  //-------------------------------------------------------------------------------------------------
  // XTS Environment; ProcessingUnit, Part, Track, Mover
  //  - instances are initialized by getting OTCIDs
  //-------------------------------------------------------------------------------------------------
  _nXpu                       : UINT := 1;  // input property in case of multiple XPU in project
  _nGroup                     : UINT;       // input property in case of multiple Xpu in project

  _nTrack                     : UINT := 1;  // this example is intended for one track only

  {attribute 'displaymode':='hex'}
  _CaGroupOID                 : OTCID; // input property frome cyclic CA group interface, MUST be set in order to do successful INIT

  // checked and evaluated in XpuCheckCycle()
  _bAllPositionsValid,
  _bMoverIdDetectionValid,
  _bMoverIdDetectionError     : BOOL;

  _nDetectedMoverCount,
  _nExpectedMoverCount        : UINT;

  _XpuOperationMode           : OperationMode;
  _MoverIdDetectionMode       : MoverIdDetectionMode;

  // XTS_Utility connection to TcCOM Object
  _fbEnvironment              : Tc3_XTS_Utility.FB_TcIoXtsEnvironment;

  // local instances of members of Environment
  // local members are connected to TcCOM by XpuInit()
  _fbProcessingUnit           : Tc3_XTS_Utility.FB_TcIoXtsProcessingUnit;

  _fbXpuPart                  : Tc3_XTS_Utility.FB_TcIoXtsXpuPart;
  _fbXpuTrack                 : Tc3_XTS_Utility.FB_TcIoXtsXpuTrack;

  _fbMc2CaGroup               : Tc3_XTS_Utility.FB_Mc2CaGroup;

  _fbPartModules              : ARRAY[1..MAX_MODULE]  OF Tc3_XTS_Utility.FB_TcIoXtsPartModule;
  _fbMoverXpu                 : ARRAY[1..MAX_MOVER]   OF Tc3_XTS_Utility.FB_TcIoXtsXpuMover;

  // TcCOM ObjectId (who am I talking to?)
  {attribute 'displaymode':='hex'}
  _Xpu_OTCID                  : OTCID;
  {attribute 'displaymode':='hex'}
  _Group_OTCID                : ARRAY[1..MAX_GROUP]   OF OTCID; // OTCID read from XPU
  {attribute 'displaymode':='hex'}
  _Part_OTCID                 : ARRAY[1..MAX_PART]    OF OTCID;
  {attribute 'displaymode':='hex'}
  _Track_OTCID                : ARRAY[1..MAX_TRACK]   OF OTCID;
  {attribute 'displaymode':='hex'}
  _Mov_OTCID                  : ARRAY[1..MAX_MOVER]   OF OTCID;
  {attribute 'displaymode':='hex'}
  _Module_OTCID               : ARRAY[1..MAX_MODULE]  OF OTCID;

  // COE Data access
  _ModuleInfoData             : REFERENCE TO ARRAY[1..MAX_MODULE] OF Tc3_XTS_Utility.ST_InfoDataView;
  _bModulePower               : ARRAY[1..MAX_MODULE] OF BOOL;

  // double check RailLength, XpuInit() will get stuck in error if not configured correctly
  _RailLengthXpu              : LREAL;
  _RailLengthGroup            : LREAL;

  _nLengthXpu,
  _nLengthGroup               : UINT;

  _nInfoServerCount,
  _nIfoStationCount,
  _nPartCount,
  _nTrackCount,
  _nTaskCount,
  _nMoverCount,
  _nModuleCount,
  _nCheckMovOID,
  _nCheckModAdr               : UINT;

  _ix                         : UINT;

  {attribute 'hide'}
  _XpuInfo                    : ST_XPU_INFO;
END_VAR

// get DcLink information from motor modules
PROPERTY AllModulesDcLink : bool
GET
VAR
  _bTmp     : BOOL;
  _nModule  : UINT;
END_VAR
IF NOT (_eInit = E_XPU_INIT.INIT_DONE) THEN RETURN; END_IF

FOR _nModule := 1 TO _nModuleCount
DO
  IF NOT _bModulePower[_nModule] // information comes from cyclic call in Cycle(): ModuleInfoData()
  THEN
    _bTmp  := FALSE;
    EXIT;
  ELSE
    _bTmp  := TRUE;
  END_IF
END_FOR

AllModulesDcLink := _bTmp;
END_GET
END_PROPERTY

PROPERTY CaGroupOID : OTCID
SET
// Group OTCID must come from the CA Group mapping in NC.Objects
_CaGroupOID := CaGroupOID;
END_SET
END_PROPERTY

METHOD Cycle : E_PROGRESS
VAR_INPUT
  Enable      : BOOL; // enable to do cyclic checks on Environment and its members
END_VAR
VAR_IN_OUT
  _eChk       : E_XPU_CHECK;
END_VAR
VAR_INST

  _eJobResult,
  _eResult      : E_PROGRESS;
  _eState       : E_PROGRESS := E_PROGRESS.PROGRESS_INIT;

END_VAR
IF NOT Enable
THEN
  ModuleInfoData(FALSE);

  _eResult  :=
  _eState   := E_PROGRESS.PROGRESS_INIT; 
  _eChk     := E_XPU_CHECK.INIT_CHECK;
END_IF 
//-----------------------------------------------------------------------------
// cyclic data fetch from Environment, ProcessingUnit, Part, ...
//-----------------------------------------------------------------------------
CASE _eState
OF
  E_PROGRESS.PROGRESS_INIT:
    IF Enable
    THEN
      _eState := _eResult         := E_PROGRESS.PROGRESS_BUSY;
    END_IF

  //---------------------------------------------------------------------------
  E_PROGRESS.PROGRESS_BUSY:       // get data from Xpu, ProcessingUnit, Part, XpuCaGroup
    _eState                       := E_PROGRESS.PROGRESS_STARTUP;

    _bAllPositionsValid           := _fbProcessingUnit.GetAreAllPositionsValid();
    _nDetectedMoverCount          := TO_UINT(_fbProcessingUnit.GetDetectedMoverCount());
    _nExpectedMoverCount          := TO_UINT(_fbProcessingUnit.GetExpectedMoverCount());
  
    _XpuOperationMode             := _fbProcessingUnit.GetOperationMode();
    _MoverIdDetectionMode         := _fbProcessingUnit.GetMoverIdDetectionMode();
  
    _RailLengthXpu                := _fbXpuPart.GetLength();
    _RailLengthGroup              := _fbMc2CaGroup.GetRailLength();
    _nLengthXpu                   := TO_UINT(_RailLengthXpu);
    _nLengthGroup                 := TO_UINT(_RailLengthGroup);
END_CASE
//-----------------------------------------------------------------------------
//-----------------------------------------------------------------------------
CASE _eState
OF
  //---------------------------------------------------------------------------
  E_PROGRESS.PROGRESS_STARTUP:    // check data for errors
    IF NOT (_bAllPositionsValid)
    THEN
      _bAllPositionsValid         := FALSE;
      _eChk                       := E_XPU_CHECK.PROCESSING_UNIT_POSITIONS_VALID;
      _eState := _eResult         := E_PROGRESS.PROGRESS_ERROR;

    ELSIF NOT (_nLengthXpu > 0)
    THEN
      _eChk                       := E_XPU_CHECK.XPU_RAIL_LENGTH;
      _eState := _eResult         := E_PROGRESS.PROGRESS_ERROR;

    ELSIF NOT (_nLengthGroup > 0)
    THEN
      _eChk                       := E_XPU_CHECK.GROUP_RAIL_LENGTH;
      _eState := _eResult         := E_PROGRESS.PROGRESS_ERROR;
     
    ELSIF NOT (_nDetectedMoverCount = _nExpectedMoverCount)
    THEN
      _bMoverIdDetectionValid     := FALSE;
      _eChk                       := E_XPU_CHECK.MOVER_COUNT_NOT_EQUAL;
      _eState := _eResult         := E_PROGRESS.PROGRESS_ERROR;
  
    ELSIF NOT (_nLengthXpu = _nLengthGroup)
    THEN
      _eChk                       := E_XPU_CHECK.RAIL_LENGTH_COMPARE;
      _eState := _eResult         := E_PROGRESS.PROGRESS_ERROR;
 
    ELSE
      _eResult                    := E_PROGRESS.PROGRESS_WORKING;

      IF NOT (__ISVALIDREF(_ModuleInfoData))
      THEN
        _eState                   := E_PROGRESS.PROGRESS_BUSY;
      ELSE
        _eJobResult               := ModuleInfoData(TRUE);
  
        IF (_eJobResult = E_PROGRESS.PROGRESS_DONE)
        THEN
          _eState                 := E_PROGRESS.PROGRESS_BUSY;
        END_IF  
      END_IF
    END_IF
END_CASE

Cycle                             := _eResult;
END_METHOD

METHOD GetEnvironment : I_TcIoXtsEnvironment
VAR_INPUT
END_VAR
GetEnvironment := _fbEnvironment;
END_METHOD

// mothers' little helper for display in visu
METHOD IdDetectionModeToString : string(20)
VAR
  _DetectionMode    : MoverIdDetectionMode; // Mover ID detection procedure
END_VAR
// just a little helper for visu display
IF NOT (_eInit = E_XPU_INIT.INIT_DONE) THEN IdDetectionModeToString := 'INIT required'; RETURN; END_IF

_DetectionMode := _fbProcessingUnit.GetMoverIdDetectionMode();

CASE _DetectionMode
OF
  MoverIdDetectionMode.Standard:
    IdDetectionModeToString       := 'Standard';

  MoverIdDetectionMode.Mover1:
    IdDetectionModeToString       := 'Mover 1';

  MoverIdDetectionMode.MultipleMover1:
    IdDetectionModeToString       := 'Multiple Mover 1';

ELSE
    IdDetectionModeToString       := 'UNKNOWN Mode';
END_CASE
END_METHOD

// mothers' little helper for display in visu
METHOD ModuleInfoData : E_PROGRESS
VAR_INPUT
  Enable        : BOOL; // enable to read ST_InfoDataView for diag/display
END_VAR
VAR_INST
  _idt,
  _nModule : UINT;
  _eReturn,
  _eState       : E_PROGRESS;
  _aPcbTemp     : ARRAY[1..4] OF REAL;
END_VAR
//---------------------------------------------------------------------------------------------
// just a little helper for visu display
// collects module data for local data
//---------------------------------------------------------------------------------------------
IF NOT (_eInit = E_XPU_INIT.INIT_DONE)      // if Xpu init is not done, just leave
THEN 
  RETURN; 
END_IF
//---------------------------------------------------------------------------------------------
IF NOT Enable                               // clear states on request
THEN
  _eReturn                                  := 
  _eState                                   := E_PROGRESS.PROGRESS_INIT; 
END_IF 
//---------------------------------------------------------------------------------------------
IF NOT (__ISVALIDREF(_ModuleInfoData))      // datafield not connected, error and leave
THEN
  ModuleInfoData                            := E_PROGRESS.PROGRESS_ERROR;
  RETURN;
END_IF
//---------------------------------------------------------------------------------------------
CASE _eState                                // get InfoData from motor modules
OF
  //-------------------------------------------------------------------------------------------
  E_PROGRESS.PROGRESS_INIT:
    IF Enable
    THEN
      _eState                                             := E_PROGRESS.PROGRESS_BUSY;
      _nModule                                            := 1;
    END_IF
END_CASE
CASE _eState
OF
  //-------------------------------------------------------------------------------------------
  E_PROGRESS.PROGRESS_BUSY:
    _eState                                               := E_PROGRESS.PROGRESS_PREPARE;

    _ModuleInfoData[_nModule].fAuxiliaryVoltage_5V        := _fbPartModules[_nModule].GetAuxiliaryVoltage5V();
    _ModuleInfoData[_nModule].fAuxiliaryVoltage_10V       := _fbPartModules[_nModule].GetAuxiliaryVoltage10V();
    _ModuleInfoData[_nModule].fAuxiliaryVoltage_24V       := _fbPartModules[_nModule].GetAuxiliaryVoltage24V();

    _ModuleInfoData[_nModule].fDcLinkVoltage              := _fbPartModules[_nModule].GetDCLinkVoltage();

    IF (_ModuleInfoData[_nModule].fDcLinkVoltage > 48.0*0.85) AND
       (_ModuleInfoData[_nModule].fDcLinkVoltage < 48.0*1.15)
    THEN
      _bModulePower[_nModule]                             := TRUE;
    ELSE
      _bModulePower[_nModule]                             := SEL((_XpuOperationMode = OperationMode.Simulation), FALSE, TRUE);
    END_IF

    _ModuleInfoData[_nModule].nCurrentScaling             := TO_INT(_fbPartModules[_nModule].GetCurrentScaling());

    _ModuleInfoData[_nModule].nDeviceInfo                 := _fbPartModules[_nModule].GetDeviceInfo();

    IF (_XpuOperationMode = OperationMode.Normal)
    THEN
      _ModuleInfoData[_nModule].fAverageTemp              := 0.0;
  
      _aPcbTemp                                           := _fbPartModules[_nModule].GetPCBTemperatures();
  
      _ModuleInfoData[_nModule].fPcbTemp_0                := _aPcbTemp[1];
      _ModuleInfoData[_nModule].fPcbTemp_1                := _aPcbTemp[2];
      _ModuleInfoData[_nModule].fPcbTemp_2                := _aPcbTemp[3];
      _ModuleInfoData[_nModule].fPcbTemp_3                := _aPcbTemp[4];

      FOR _idt := 1 TO 4
      DO
        _ModuleInfoData[_nModule].fAverageTemp            := _ModuleInfoData[_nModule].fAverageTemp + _aPcbTemp[_idt];
      END_FOR
      _ModuleInfoData[_nModule].fAverageTemp              := _ModuleInfoData[_nModule].fAverageTemp / 4;
    END_IF

    _ModuleInfoData[_nModule].fOverallCurrent             := _fbPartModules[_nModule].GetOverallCurrent();

    _ModuleInfoData[_nModule].fMaxDCLinkVoltageLast500ms  := _fbPartModules[_nModule].GetMaxDCLinkVoltageLast500ms();
    _ModuleInfoData[_nModule].fMaxOverallCurrentLast500ms := _fbPartModules[_nModule].GetMaxOverallCurrentLast500ms();
END_CASE
CASE _eState 
OF
  //-------------------------------------------------------------------------------------------
  E_PROGRESS.PROGRESS_PREPARE:
    IF (_nModule > _nModuleCount-1)
    THEN
      _eState                                             := E_PROGRESS.PROGRESS_WORKING;
    ELSE
      _nModule                                            := _nModule + 1;
      _eReturn                                            :=
      _eState                                             := E_PROGRESS.PROGRESS_BUSY;
    END_IF

  //-------------------------------------------------------------------------------------------
  E_PROGRESS.PROGRESS_WORKING:
    _eReturn                                              := E_PROGRESS.PROGRESS_DONE;
    _eState                                               := E_PROGRESS.PROGRESS_INIT;
END_CASE

ModuleInfoData                                            := _eReturn;
END_METHOD

// mothers' little helper for display in visu
METHOD MoverPositionAssignementToString : string(20)
VAR
  _PositionAssignement    : MoverPositionAssignment; // XPU movver assignement procedure
END_VAR
// just a little helper for visu display
IF NOT (_eInit = E_XPU_INIT.INIT_DONE) THEN MoverPositionAssignementToString := 'INIT required'; RETURN; END_IF

_PositionAssignement      := _fbProcessingUnit.GetMoverPositionAssignment();

CASE _PositionAssignement
OF
  MoverPositionAssignment.Standard:
    MoverPositionAssignementToString    := 'Standard';

  MoverPositionAssignment.StartAtFirstMover:
    MoverPositionAssignementToString    := 'Start At First Mover';
ELSE
    MoverPositionAssignementToString    := 'UNKNOWN Assgnement';
END_CASE
END_METHOD

// mothers' little helper for display in visu
METHOD OpModeToString : String(20)
VAR
  _OpMode     : OperationMode; // XPU operation mode
END_VAR
// just a little helper for visu display
IF NOT (_eInit = E_XPU_INIT.INIT_DONE) THEN OpModeToString := 'INIT required'; RETURN; END_IF

_OpMode   := _fbProcessingUnit.GetOperationMode();

CASE _OpMode
OF
  OperationMode.Normal:
    OpModeToString      := 'Normal';

  OperationMode.Simulation:
    OpModeToString      := 'Simulation';

ELSE
    OpModeToString      := 'UNKNOWN OP MODE';
END_CASE
END_METHOD

PROPERTY RailLength : lreal
GET
IF (_eInit = E_XPU_INIT.INIT_DONE)
THEN
  RailLength := _fbXpuPart.GetLength();
ELSE
  RailLength := 0.0;
END_IF
END_GET
END_PROPERTY

PROPERTY XpuInfo : st_xpu_info
GET
IF NOT (_eInit = E_XPU_INIT.INIT_DONE) THEN RETURN; END_IF

_XpuInfo.AllPositionsValid        := _bAllPositionsValid;

_XpuInfo.IdDetectionError         := _bMoverIdDetectionError;
_XpuInfo.IdDetectionValid         := _bMoverIdDetectionValid;

_XpuInfo.IdDetectionActive        := _fbProcessingUnit.GetIsMoverIdDetectionActive();

_XpuInfo.OperationMode            := TO_UINT(_fbProcessingUnit.GetOperationMode());

_XpuInfo.IdDetectionMode          := TO_UINT(_fbProcessingUnit.GetMoverIdDetectionMode());
_XpuInfo.MoverPositionAssignement := TO_UINT(_fbProcessingUnit.GetMoverPositionAssignment());

_XpuInfo.nDetectedAxisCount       := _nDetectedMoverCount;
_XpuInfo.nExpectedAxisCount       := _nExpectedMoverCount;

XpuInfo := _XpuInfo;
END_GET
END_PROPERTY

METHOD XpuInit  : E_XPU_INIT      // connect to TcCOM
VAR_INPUT
  Execute       : BOOL;           // must be executed for connecting to TcCOM Environment of Xpu
END_VAR
VAR_IN_OUT
  _eReslt       : E_PROGRESS;     // send info about progress to caller
  _eChk         : E_XPU_CHECK;
END_VAR
VAR_INST
  _eState         : E_PROGRESS;   // progress state
  _nState         : E_XPU_INIT;   // initialization state
  _eDataGetCount  : E_PROGRESS;   // cycle counter to catch exceeding wait time for data from ProcessingUnit
END_VAR
// clear progress on request
IF NOT Execute 
THEN 
  _eState                           := E_PROGRESS.PROGRESS_INIT;
  _eDataGetCount                    := 0;
 
  XpuInit                           :=
  _nState                           := E_XPU_INIT.INIT_START; 
  RETURN; 
END_IF

// progress state
CASE _eState
OF
  E_PROGRESS.PROGRESS_INIT:         // clear start
    IF Execute
    THEN
      _eState                       := E_PROGRESS.PROGRESS_BUSY;
      _eChk                         := E_XPU_CHECK.INIT_CHECK;    // clear cyclic check state

      // always initialize environment function blocks to get defined start of progress
      _fbEnvironment.Init(FALSE);
      _fbEnvironment.GetXpuOids(FALSE);
      _fbEnvironment.GetInfoServerOids(FALSE);

      // clear initialization states
      _nState                       := E_XPU_INIT.INIT_START;

      // clear check bits
      _bAllPositionsValid           :=
      _bMoverIdDetectionValid       :=
      _bMoverIdDetectionError       := FALSE;

      // clear check values
      _nLengthXpu                   :=
      _nLengthGroup                 :=
      _nDetectedMoverCount          :=
      _nExpectedMoverCount          := 0;

      // clear work values
      _nInfoServerCount             :=
      _nIfoStationCount             :=
      _nPartCount                   :=
      _nTrackCount                  :=
      _nTaskCount                   :=
      _nMoverCount                  :=
      _nModuleCount                 :=
      _nCheckMovOID                 :=
      _nCheckModAdr                 := 0;
    END_IF
END_CASE
//-----------------------------------------------------------------------------
//-----------------------------------------------------------------------------
CASE _eState
OF
  E_PROGRESS.PROGRESS_BUSY:         // begin with initializing environment
    CASE _nState
    OF
    INIT_START:                     // call initialization of environment
      _fbEnvironment.Init(TRUE);

      // get information about success in Property (P_<function>)
      IF _fbEnvironment.P_IsInitialized
      THEN
        // now environment is fully initialized
        // access to members by use of provided interfaces
        // if you use interfaces, things are done here (change to your needs.., rewrite this section...)
        //------------------------------------------------------------------------------------------------
        
        //---------------------------------------------------------------------
        // use of local function block instances
        // get information about Object IDs to local datafields
        //---------------------------------------------------------------------
        //  - everything else in this state machine is for use within fb_Xpu
        //  - the following states shall illustrate how TcCOM Objects are connected through XTS_Utility lib
        //  - local instances of members of Environment are connected from here onward
        //
        IF _fbEnvironment.GetXpuOids(TRUE) // get object IDs for all processing units
        THEN
          _fbEnvironment.Init(FALSE);// clear environment init
          _nState                   := INIT_ENVIRONMENT_OID;
        END_IF
      END_IF

    INIT_ENVIRONMENT_OID:           // get processing unit object ID for THIS instance
      _Xpu_OTCID                    := _fbEnvironment.P_XpuOids[_nXpu];   // fb_Xpu.XpuInstance --> _nXpu

      // clear all local object IDs
      memset(ADR(_Part_OTCID)    , 0, SIZEOF(_Part_OTCID));
      memset(ADR(_Track_OTCID)   , 0, SIZEOF(_Track_OTCID));
      memset(ADR(_Mov_OTCID)     , 0, SIZEOF(_Mov_OTCID));
      memset(ADR(_Module_OTCID)  , 0, SIZEOF(_Module_OTCID));

      // clear function blocks
      _fbEnvironment.GetXpuOids     (FALSE);
      _fbEnvironment.GetCaGroupCount(FALSE);
      _fbEnvironment.GetInfoServerCount(FALSE);

      _nState                       := INIT_INFO_SERVER_ITF;              // check environment for info servers

    INIT_INFO_SERVER_ITF:           // HAUD 2024 03 14: TODO - implement procedure for getting Info server data to local datafields
      IF _fbEnvironment.GetInfoServerCount(TRUE)
      THEN
        // how many of you are there?
        _nInfoServerCount           := _fbEnvironment.P_InfoServerCount;

        IF (_nInfoServerCount > 0)
        THEN
          // go do something with the data
          //
          //  TODO - get station coordinates
          _eState                   := E_PROGRESS.PROGRESS_PREPARE; // TODO - implement InfoServer R/W
          _nState                   := INIT_CA_GROUP_OID;           // TODO - implement initialization states for info server procedure

        ELSE
          // no info server present
          _eState                   := E_PROGRESS.PROGRESS_PREPARE;
          _nState                   := INIT_CA_GROUP_OID; // go check CA group
        END_IF
      END_IF
    END_CASE
END_CASE
//-----------------------------------------------------------------------------
//-----------------------------------------------------------------------------
CASE _eState
OF
  E_PROGRESS.PROGRESS_PREPARE:      // CA group initialization
    CASE _nState
    OF
    INIT_CA_GROUP_OID:              // get object IDs of all CA groups in environment
      IF _fbEnvironment.GetCaGroupOids(TRUE)
      THEN
        _Group_OTCID                := _fbEnvironment.P_CaGroupOids;  // copy all Ids to local
        _nState                     := INIT_CA_GROUP_GET_OID;
      END_IF

    INIT_CA_GROUP_GET_OID:          // look for any CA group
      _fbEnvironment.GetCaGroupOids(FALSE);
      IF NOT (_Group_OTCID[1] <> 0)
      THEN
        // no group is configured in project --> error, go add/link CA Group in NC objects
        _eChk                       := E_XPU_CHECK.GROUP_NOT_CONFIGURED;
        _eState                     := E_PROGRESS.PROGRESS_ERROR;
      ELSE
        _nState                     := INIT_CA_GROUP_CHECK_OID; // get matching CA group
      END_IF

    INIT_CA_GROUP_CHECK_OID:        // ID must be found, there is one chance
      _eChk                         := E_XPU_CHECK.GROUP_OID_MISMATCH;
      _eState                       := E_PROGRESS.PROGRESS_ERROR;

      FOR _ix := 1 TO MAX_GROUP
      DO
        IF (_fbEnvironment.P_CaGroupOids[_ix] <> 0)
        THEN
          // check whether the input from cyclic interface can be found in XPU data
          IF (_fbEnvironment.P_CaGroupOids[_ix] = _CaGroupOID)  // _CaGroupOID must be linked from NC Objects into PLC (GROUP_REF)
          THEN

            _eState                 := E_PROGRESS.PROGRESS_PREPARE;
            _eChk                   := E_XPU_CHECK.INIT_CHECK;

            _nGroup                 := _ix;

            _fbEnvironment.GetCaGroupOids(FALSE);
            _nState                 := INIT_CA_GROUP_COM; // only continue if match was found
            EXIT;
          END_IF
        END_IF
      END_FOR

    INIT_CA_GROUP_COM:              // connect to CaGroup function block in environment
      IF (_fbMc2CaGroup.GetComObject(_fbEnvironment.P_CaGroupOids[_nGroup]))
      THEN
        _eState                     := E_PROGRESS.PROGRESS_STARTUP;
        _nState                     := INIT_PROCESSING_UNIT_COM;
      END_IF
    END_CASE
END_CASE
//-----------------------------------------------------------------------------
//-----------------------------------------------------------------------------
CASE _eState
OF
  E_PROGRESS.PROGRESS_STARTUP:      // ProcessingUnit initialization
  CASE _nState
  OF
  INIT_PROCESSING_UNIT_COM:         // connect local function block with TcCom object
    IF (_fbProcessingUnit.GetComObject(_Xpu_OTCID))
    THEN
      // local function block can now be used to get information
      // get operation mode first
      _XpuOperationMode             := _fbProcessingUnit.GetOperationMode();
      _nState                       := INIT_PROCESSING_UNIT_PART_COUNT;
    END_IF

  INIT_PROCESSING_UNIT_PART_COUNT:  // get parts in ProcessingUnit
    _nPartCount                     := TO_UINT(_fbProcessingUnit.GetPartCount());

    IF (_nPartCount > 0)            // one is enough
    THEN
      _nState                       := INIT_PROCESSING_UNIT_PART_OID;
    END_IF

  INIT_PROCESSING_UNIT_PART_OID:    // get object IDs of all parts in ProcessingUNit
    IF _fbProcessingUnit.GetPartOids()
    THEN
      _eState                       := E_PROGRESS.PROGRESS_CHECK;

      _Part_OTCID                   := _fbProcessingUnit.P_PartOids;  // copy IDs to local
      _nState                       := INIT_PROCESSING_UNIT_TRACK_COUNT;
    END_IF
  END_CASE
END_CASE
//-----------------------------------------------------------------------------
//-----------------------------------------------------------------------------
CASE _eState
OF
  E_PROGRESS.PROGRESS_CHECK:        // track initialization
  CASE _nState
  OF
  INIT_PROCESSING_UNIT_TRACK_COUNT: // how many tracks does this ProcessingUnit have?
    _nTrackCount                    := TO_UINT(_fbProcessingUnit.GetTrackCount());
  
    IF (_nTrackCount > 0)           // one is enough
    THEN
      _nState                       := INIT_PROCESSING_UNIT_TRACK_OID;
    END_IF

  INIT_PROCESSING_UNIT_TRACK_OID:   // get object IDs of all tracks in ProcessingUnit
    IF _fbProcessingUnit.GetTrackOids()
    THEN
      _eState                       := E_PROGRESS.PROGRESS_OCCUPIED;

      _Track_OTCID                  := _fbProcessingUnit.P_TrackOids; // copy IDs to local
      _nState                       := INIT_PROCESSING_UNIT_MOVER_COUNT;
    END_IF
  END_CASE
END_CASE
//-----------------------------------------------------------------------------
//-----------------------------------------------------------------------------
CASE _eState
OF
  E_PROGRESS.PROGRESS_OCCUPIED:     // Mover initialization
  CASE _nState
  OF
  INIT_PROCESSING_UNIT_MOVER_COUNT: // how many of you are there?
    _nMoverCount                    := TO_UINT(_fbProcessingUnit.GetMoverCount());
  
    IF (_nMoverCount > 0)           // one is enough
    THEN
      _nState                       := INIT_PROCESSING_UNIT_MOVER_OID;
    END_IF

  INIT_PROCESSING_UNIT_MOVER_OID:   // get object IDs of all mover in ProcessingUnit
    IF _fbProcessingUnit.GetMoverOids()
    THEN
      _eState                       := E_PROGRESS.PROGRESS_WORKING;

      _Mov_OTCID                    := _fbProcessingUnit.P_MoverOids; // copy IDs to local
      _nState                       := INIT_PROCESSING_UNIT_TASK_COUNT;
      _eChk                         := E_XPU_CHECK.MOVER_COUNT;
    END_IF
  END_CASE
END_CASE
//-----------------------------------------------------------------------------
//-----------------------------------------------------------------------------
CASE _eState
OF
  E_PROGRESS.PROGRESS_WORKING:      // task information
  CASE _nState
  OF
  INIT_PROCESSING_UNIT_TASK_COUNT:  // how many?
    _nTaskCount                     := TO_UINT(_fbProcessingUnit.GetTaskCount());
  
    IF (_nTaskCount > 0)
    THEN
      _nState                       := INIT_PROCESSING_UNIT_TASK_OID;
    END_IF    

  INIT_PROCESSING_UNIT_TASK_OID:    // get their names!
    IF _fbProcessingUnit.GetTaskOids()
    THEN
      _eState                       := E_PROGRESS.PROGRESS_STILL_WORKING;
      _nState                       := INIT_TRACK_COM;
    END_IF
  END_CASE
END_CASE
//-----------------------------------------------------------------------------
//-----------------------------------------------------------------------------
CASE _eState
OF
  E_PROGRESS.PROGRESS_STILL_WORKING:// connect local instances of track, part, modules and mover
    CASE _nState
    OF
    INIT_TRACK_COM:                 // get TcCom Object for my track (_nTrack is fixed to 1 in this example; multi track is not intended)
      IF _fbXpuTrack.GetComObject(_Track_OTCID[_nTrack])
      THEN
        _nState                     := INIT_PART_COM;
      END_IF
    //-----------------------------------------------------------------------------------------------
    //-----------------------------------------------------------------------------------------------
    INIT_PART_COM:                  // get TcCom object for my part (also fixed to 1 part per ProcessingUnit; multi part is not intended)
      IF _fbXpuPart.GetComObject(_Part_OTCID[1])
      THEN
        _nState                     := INIT_PART_MODULE_COUNT;
      END_IF
    //-----------------------------------------------------------------------------------------------
    //-----------------------------------------------------------------------------------------------
    INIT_PART_MODULE_COUNT:         // get count of motor modules
      _nModuleCount                 := TO_UINT(_fbXpuPart.GetModuleCount());
    
      IF (_nModuleCount > 0)        // one is enough
      THEN
        _nState                     := INIT_PART_MODULE_OID;
      END_IF
    //-----------------------------------------------------------------------------------------------
    //-----------------------------------------------------------------------------------------------
    INIT_PART_MODULE_OID:           // get object IDs of all motor modules in part
      IF _fbXpuPart.GetModuleOids()
      THEN
        _Module_OTCID               := _fbXpuPart.P_ModuleOids; // copy IDs to local
    
        _nState                     := INIT_PART_MODULE_COM;    // go, connect module IDs
        _nCheckModAdr               := 1;                       // start at first module
      END_IF
    //-----------------------------------------------------------------------------------------------
    //-----------------------------------------------------------------------------------------------
    INIT_PART_MODULE_COM:           // connect to TcCom object
      IF _fbPartModules[_nCheckModAdr].GetComObject(_Module_OTCID[_nCheckModAdr])
      THEN
        _nState                     := INIT_PART_MODULE_COM_NEXT;
      END_IF
    //-----------------------------------------------------------------------------------------------
    INIT_PART_MODULE_COM_NEXT:
      IF (_nCheckModAdr > _nModuleCount-1)
      THEN
        // all data from modules collected, continue to mover data
        _nState                     := INIT_MOVER_COM;          // go, connect mover IDs 
        _nCheckMovOID               :=  1;                      // start at first mover
      ELSE
        // still data to fetch, increment search index, go back to fetching data
        _nState                     := INIT_PART_MODULE_COM;    // go back for next
        _nCheckModAdr               := _nCheckModAdr + 1;       // next
      END_IF
    //-----------------------------------------------------------------------------------------------
    //-----------------------------------------------------------------------------------------------
    INIT_MOVER_COM:                 // connect to TcCom object
      IF _fbMoverXpu[_nCheckMovOID].GetComObject(_Mov_OTCID[_nCheckMovOID])
      THEN
        _nState                     := INIT_MOVER_COM_NEXT;
      END_IF
    //-----------------------------------------------------------------------------------------------
    INIT_MOVER_COM_NEXT:
      IF (_nCheckMovOID > _nMoverCount-1)
      THEN
        // all done
        _nState                     := INIT_DATA_GET;           // get important data from ProcessingUnit etc...
      ELSE
        // more data to fetch, increment search index and go back
        _nState                     := INIT_MOVER_COM;          // go back for next
        _nCheckMovOID               := _nCheckMovOID + 1;       // next
      END_IF
    //-----------------------------------------------------------------------------------------------
    //-----------------------------------------------------------------------------------------------
    INIT_DATA_GET:                  // get data, add more if your application requires it
      // start counter
      _eDataGetCount                := _eDataGetCount + 1;
      IF (_eDataGetCount MOD E_PROGRESS.PROGRESS_ERROR = 0)
      THEN
        _eState                     := E_PROGRESS.PROGRESS_ERROR;
        _eCheck                     := E_XPU_CHECK.PROCESSING_UNIT_GET_DATA_EXCEED;
      END_IF
      // wait for plausible data from members
      IF (_bAllPositionsValid) AND
         (_nLengthXpu > 0)
      THEN
        _nState                     := INIT_DATA_CHECK;
        _eChk                       := E_XPU_CHECK.PROCESSING_UNIT_POSITIONS_VALID;
      END_IF

      _bAllPositionsValid           := _fbProcessingUnit.GetAreAllPositionsValid();
      _nDetectedMoverCount          := TO_UINT(_fbProcessingUnit.GetDetectedMoverCount());
      _nExpectedMoverCount          := TO_UINT(_fbProcessingUnit.GetExpectedMoverCount());

      _XpuOperationMode             := _fbProcessingUnit.GetOperationMode();
      _MoverIdDetectionMode         := _fbProcessingUnit.GetMoverIdDetectionMode();

      _RailLengthXpu                := _fbXpuPart.GetLength();
      _RailLengthGroup              := _fbMc2CaGroup.GetRailLength();
      _nLengthXpu                   := TO_UINT(_RailLengthXpu);
      _nLengthGroup                 := TO_UINT(_RailLengthGroup);

    //-----------------------------------------------------------------------------------------------
    INIT_DATA_CHECK:                // plausibility checks
      IF NOT (_nDetectedMoverCount = _nExpectedMoverCount)
      THEN
        _eChk                       := E_XPU_CHECK.MOVER_COUNT_NOT_EQUAL; // the thing that must not be
        _eState                     := E_PROGRESS.PROGRESS_ERROR;

      ELSIF NOT (_nLengthXpu = _nLengthGroup)
      THEN
        _eChk                       := E_XPU_CHECK.RAIL_LENGTH_COMPARE;   // yet another thing that must not be
        _eState                     := E_PROGRESS.PROGRESS_ERROR;

      ELSE
        _nState                     := INIT_DONE;                         // write success
      END_IF
    //-----------------------------------------------------------------------------------------------
    INIT_DONE:
      _eState                       := E_PROGRESS.PROGRESS_DONE;          // method is done
    END_CASE
END_CASE

_eReslt                             := _eState;
XpuInit                             := _nState;
END_METHOD

PROPERTY XpuInstance : uint
SET
//
// Who am I?
// Environment may have more than one ProcessingUnit,
// information required for connecting to the correct instance of ProcessingUnit
_nXpu := XpuInstance;
END_SET
END_PROPERTY

PROPERTY XpuModuleInfoData : REFERENCE TO ARRAY[1..MAX_MODULE] OF Tc3_XTS_Utility.ST_InfoDataView
SET

_ModuleInfoData REF= XpuModuleInfoData;
END_SET
END_PROPERTY

END_FUNCTION_BLOCK

// ---- XTS/_Visualization/MOVER_VISU.TcVIS
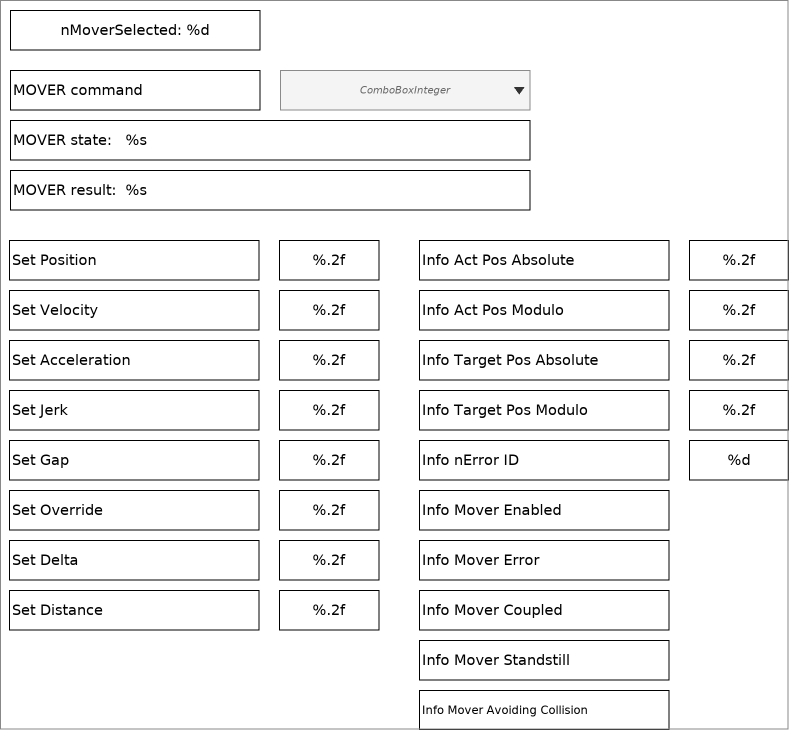
VISUALIZATION MOVER_VISU  // 789x730
    Rectangle (10,10 250x40), "nMoverSelected: %d", text variable: MAIN.nMoverSelected
        OnMouseClick: write the text variable via VisuDialogs.Numpad, min 1, max MAX_MOVER, title 'Selected Mover'
    Rectangle (10,120 520x40), "MOVER state: %s", text variable: MAIN.sMoverState
    Rectangle (10,70 250x40), "MOVER command"
    ComboBoxInteger (280,70 250x40), variable: GVL_XTS.MoverCtrl[MAIN.nMoverSelected].Cmd, text list: 'TL_E_CTRL_MOVER'
    Rectangle (10,170 520x40), "MOVER result: %s", text variable: MAIN.sMoverResult
    Rectangle (9,240 250x40), "Set Position"
    Rectangle (9,290 250x40), "Set Velocity"
    Rectangle (9,340 250x40), "Set Acceleration"
    Rectangle (9,390 250x40), "Set Jerk"
    Rectangle (9,440 250x40), "Set Gap"
    Rectangle (9,490 250x40), "Set Override"
    Rectangle (9,540 250x40), "Set Delta"
    Rectangle (9,590 250x40), "Set Distance"
    Rectangle (279,240 100x40), "%.2f", text variable: GVL_XTS.MoveData[MAIN.nMoverSelected].rPos
        OnMouseClick: write the text variable via Default
    Rectangle (279,290 100x40), "%.2f", text variable: GVL_XTS.MoveData[MAIN.nMoverSelected].rVelo
        OnMouseClick: write the text variable via Default
    Rectangle (279,340 100x40), "%.2f", text variable: GVL_XTS.MoveData[MAIN.nMoverSelected].rAcc
        OnMouseClick: write the text variable via Default
    Rectangle (279,390 100x40), "%.2f", text variable: GVL_XTS.MoveData[MAIN.nMoverSelected].rJerk
        OnMouseClick: write the text variable via Default
    Rectangle (279,440 100x40), "%.2f", text variable: GVL_XTS.MoveData[MAIN.nMoverSelected].rGap
        OnMouseClick: write the text variable via Default
    Rectangle (279,490 100x40), "%.2f", text variable: GVL_XTS.MoveData[MAIN.nMoverSelected].rOverride
        OnMouseClick: write the text variable via Default
    Rectangle (279,540 100x40), "%.2f", text variable: GVL_XTS.MoveData[MAIN.nMoverSelected].rDelta
        OnMouseClick: write the text variable via Default
    Rectangle (279,590 100x40), "%.2f", text variable: GVL_XTS.MoveData[MAIN.nMoverSelected].rDistance
        OnMouseClick: write the text variable via Default
    Rectangle (419,240 250x40), "Info Act Pos Absolute"
    Rectangle (419,290 250x40), "Info Act Pos Modulo"
    Rectangle (419,340 250x40), "Info Target Pos Absolute"
    Rectangle (419,390 250x40), "Info Target Pos Modulo"
    Rectangle (419,440 250x40), "Info nError ID"
    Rectangle (689,240 100x40), "%.2f", text variable: GVL_XTS.MoverInfo[MAIN.nMoverSelected].rAbsActPos
    Rectangle (689,290 100x40), "%.2f", text variable: GVL_XTS.MoverInfo[MAIN.nMoverSelected].rModuloActPos
    Rectangle (689,340 100x40), "%.2f", text variable: GVL_XTS.MoverInfo[MAIN.nMoverSelected].rAbsTargetPos
    Rectangle (689,390 100x40), "%.2f", text variable: GVL_XTS.MoverInfo[MAIN.nMoverSelected].rModuloTargetPos
    Rectangle (689,440 100x40), "%d", text variable: GVL_XTS.MoverInfo[MAIN.nMoverSelected].nErrorId
    Rectangle (419,490 250x40), "Info Mover Enabled", colour toggle: GVL_XTS.MoverInfo[MOVER.nMoverSelected].bMoverEnabled
    Rectangle (419,540 250x40), "Info Mover Error", colour toggle: GVL_XTS.MoverInfo[MOVER.nMoverSelected].bMoverError
    Rectangle (419,590 250x40), "Info Mover Coupled", colour toggle: GVL_XTS.MoverInfo[MOVER.nMoverSelected].bMoverCoupled
    Rectangle (419,640 250x40), "Info Mover Standstill", colour toggle: GVL_XTS.MoverInfo[MOVER.nMoverSelected].bMoverStandstill
    Rectangle (419,690 250x40), "Info Mover Avoiding Collision", colour toggle: GVL_XTS.MoverInfo[MOVER.nMoverSelected].bMoverAvoidingCollision
END_VISUALIZATION

// ---- XTS/_Visualization/textlists/TL_E_CTRL_MOVER.TcTLO
TEXTLIST TL_E_CTRL_MOVER
  0 = 'MOVER_NULL'
  1 = 'MOVER_ENABLE'
  2 = 'MOVER_DISABLE'
  4 = 'MOVER_MOVE_TO_POS_CA'
  5 = 'MOVER_SEND_TO_POS_CA'
  6 = 'MOVER_HALT'
  7 = 'MOVER_GEAR_IN'
  8 = 'MOVER_GEAR_IN_POS_CA'
  9 = 'MOVER_GEAR_OUT'
  10 = 'MOVER_RESET'
  3 = 'MOVER_MOVE_TO_POS'
   = ''
END_TEXTLIST

// ---- XTS/_Visualization/XPU_VISU.TcVIS
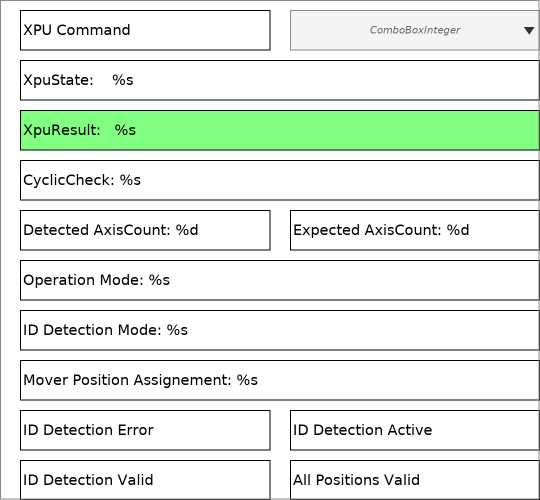
VISUALIZATION XPU_VISU  // 540x500
    Rectangle (20,10 250x40), "XPU Command"
    ComboBoxInteger (290,10 250x40), variable: GVL_XTS.XpuCtrl.Cmd, text list: 'TL_E_CTRL_XPU'
    Rectangle (20,160 520x40), "CyclicCheck: %s", text variable: MAIN.sXpuCheck
    Rectangle (20,60 520x40), "XpuState: %s", text variable: MAIN.sXpuState
    Rectangle (20,110 520x40), "XpuResult: %s", text variable: MAIN.sXpuResult, colour toggle: (MAIN.eXpuResult = E_PROGRESS.PROGRESS_ERROR)
    Rectangle (290,460 250x40), "All Positions Valid", colour toggle: GVL_XTS.XpuInfo.AllPositionsValid
    Rectangle (20,410 250x40), "ID Detection Error", colour toggle: GVL_XTS.XpuInfo.IdDetectionError
    Rectangle (20,460 250x40), "ID Detection Valid", colour toggle: GVL_XTS.XpuInfo.IdDetectionValid
    Rectangle (290,410 250x40), "ID Detection Active", colour toggle: GVL_XTS.XpuInfo.IdDetectionActive
    Rectangle (20,260 520x40), "Operation Mode: %s", text variable: MAIN.sXpuOpMode
    Rectangle (20,310 520x40), "ID Detection Mode: %s", text variable: MAIN.sXpuMoverdetectionMode
    Rectangle (20,360 520x40), "Mover Position Assignement: %s", text variable: MAIN.sXpuMoverAssignement
    Rectangle (290,210 250x40), "Expected AxisCount: %d", text variable: GVL_XTS.XpuInfo.nExpectedAxisCount
    Rectangle (20,210 250x40), "Detected AxisCount: %d", text variable: GVL_XTS.XpuInfo.nDetectedAxisCount
END_VISUALIZATION
